// Mitsubishi GX Works2 project: PLCAI   PLC: FX3U/FX3UC

PROGRAM MAIN
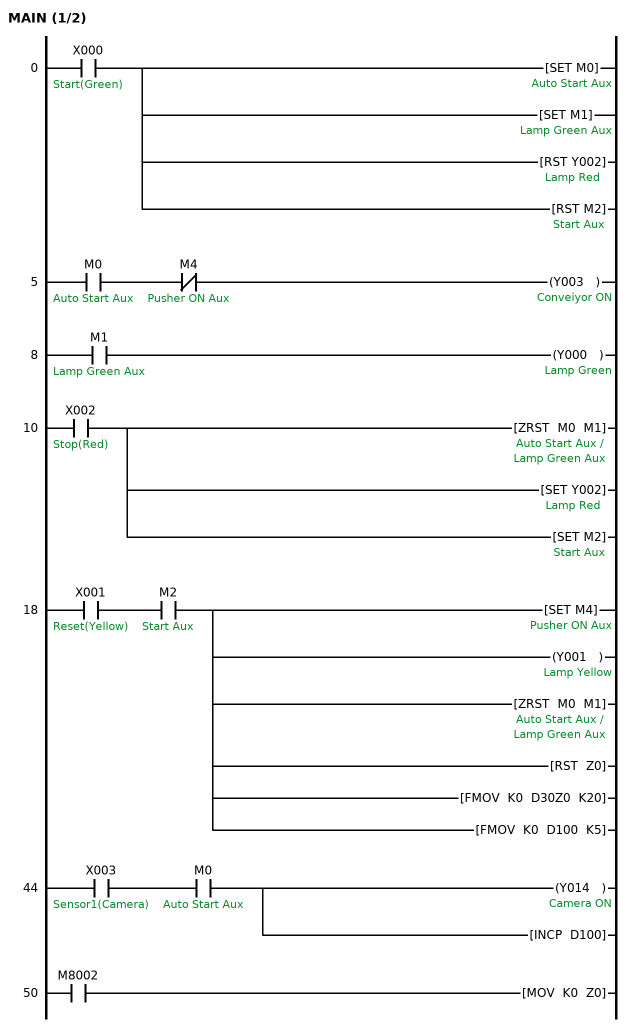
0     LD      X000  ; Start(Green)
      SET     M0  ; Auto Start Aux
      SET     M1  ; Lamp Green Aux
      RST     Y002  ; Lamp Red
      RST     M2  ; Start Aux
5     LD      M0  ; Auto Start Aux
      ANI     M4  ; Pusher ON Aux
      OUT     Y003  ; Conveiyor ON
8     LD      M1  ; Lamp Green Aux
      OUT     Y000  ; Lamp Green
10    LD      X002  ; Stop(Red)
      ZRST    M0 M1
      SET     Y002  ; Lamp Red
      SET     M2  ; Start Aux
18    LD      X001  ; Reset(Yellow)
      AND     M2  ; Start Aux
      SET     M4  ; Pusher ON Aux
      OUT     Y001  ; Lamp Yellow
      ZRST    M0 M1
      RST     Z0
      FMOV    K0 D30Z0 K20
      FMOV    K0 D100 K5
44    LD      X003  ; Sensor1(Camera)
      AND     M0  ; Auto Start Aux
      OUT     Y014  ; Camera ON
      INCP    D100
50    LD      M8002
      MOV     K0 Z0
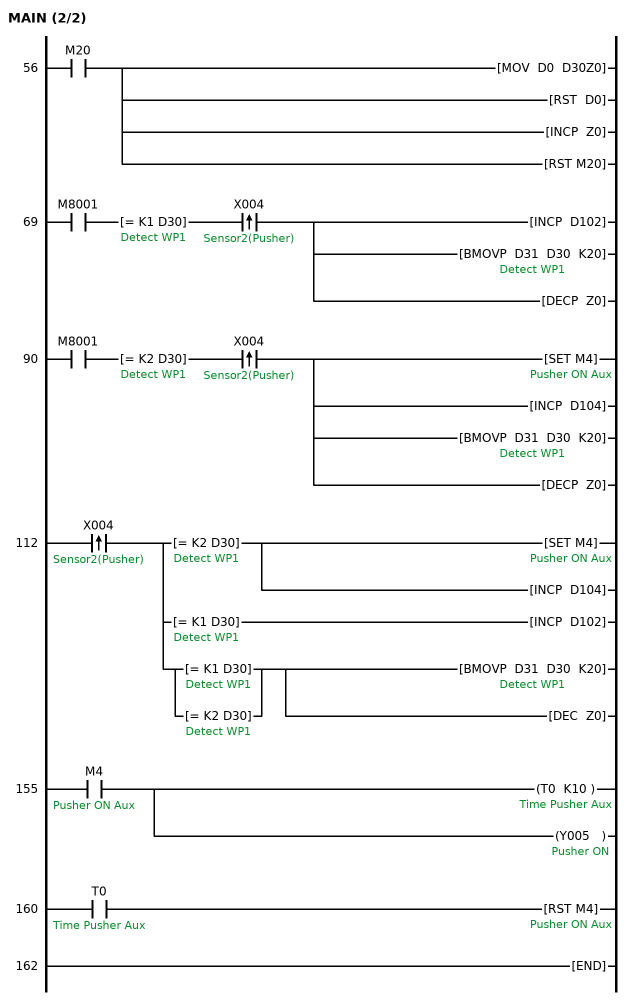
56    LD      M20
      MOV     D0 D30Z0
      RST     D0
      INCP    Z0
      RST     M20
69    LD      M8001
      AND=    K1 D30  ; Detect WP1
      ANDP    X004  ; Sensor2(Pusher)
      INCP    D102
      BMOVP   D31 D30 K20
      DECP    Z0
90    LD      M8001
      AND=    K2 D30  ; Detect WP1
      ANDP    X004  ; Sensor2(Pusher)
      SET     M4  ; Pusher ON Aux
      INCP    D104
      BMOVP   D31 D30 K20
      DECP    Z0
112   LDP     X004  ; Sensor2(Pusher)
      MPS
      AND=    K2 D30  ; Detect WP1
      SET     M4  ; Pusher ON Aux
      INCP    D104
      MRD
      AND=    K1 D30  ; Detect WP1
      INCP    D102
      MPP
      LD=     K1 D30  ; Detect WP1
      OR=     K2 D30  ; Detect WP1
      ANB
      BMOVP   D31 D30 K20
      DEC     Z0
155   LD      M4  ; Pusher ON Aux
      OUT     T0 K10  ; Time Pusher Aux
      OUT     Y005  ; Pusher ON
160   LD      T0  ; Time Pusher Aux
      RST     M4  ; Pusher ON Aux
162   END
END_PROGRAM

// device comments not shown above
M10  ; Force ON Camera
M11  ; Force ON Pusher
